# EPICS autosave request: ffmpegServer/iocs/ffmpegServerIOC/iocBoot/iocffmpegServer/auto_settings.req
file "simDetector_settings.req",    P=$(P),  R=cam1:
file "ADBase_settings.req",         P=$(P),  R=cam1:
file "NDPluginBase_settings.req",   P=$(P),  R=image1:
file "NDStdArrays_settings.req",    P=$(P),  R=image1:
file "commonPlugin_settings.req",   P=$(P)
